% RSLogix 500 project MLO3B JOb 8.RSS, saved by version 10.00.00.00 %
PROJECT "MLO3B"    % processor: Bul.1763 MicroLogix 1100 Series B %

PROGRAM FILES
  LAD 2   5 rungs

DATA FILES
  O0 OUTPUT  4 elements
  I1 INPUT  6 elements
  S2 STATUS  66 elements
  B3 BINARY  1 elements
  T4 TIMER  1 elements
  C5 COUNTER  1 elements
  R6 CONTROL  1 elements
  N7 INTEGER  1 elements
  F8 FLOAT  1 elements

LADDER 2
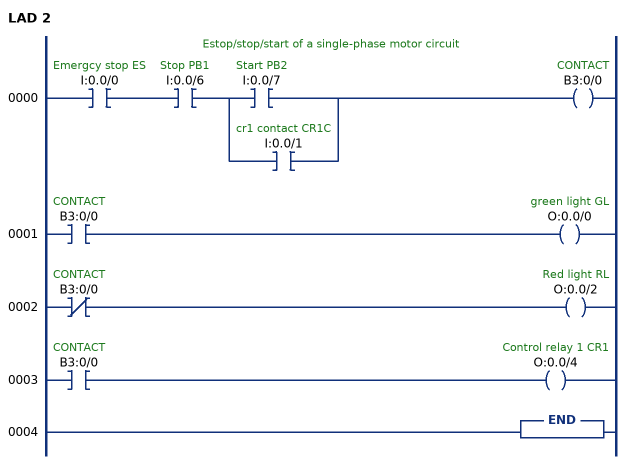
% Rung: 0 %
% Estop/stop/start of a single-phase motor circuit %
SOR XIC I:0.0/0 XIC I:0.0/6 BST XIC I:0.0/7 NXB XIC I:0.0/1 BND OTE B3:0/0 EOR
%   I:0.0/0  ES  "Emergcy stop" %
%   I:0.0/6  PB1  "Stop" %
%   I:0.0/7  PB2  "Start" %
%   I:0.0/1  CR1C  "cr1 contact" %
%   B3:0/0  CONTACT %
% Rung: 1 %
SOR XIC B3:0/0 OTE O:0.0/0 EOR
%   B3:0/0  CONTACT %
%   O:0.0/0  GL  "green light" %
% Rung: 2 %
SOR XIO B3:0/0 OTE O:0.0/2 EOR
%   B3:0/0  CONTACT %
%   O:0.0/2  RL  "Red light" %
% Rung: 3 %
SOR XIC B3:0/0 OTE O:0.0/4 EOR
%   B3:0/0  CONTACT %
%   O:0.0/4  CR1  "Control relay 1" %
% Rung: 4 %
SOR END EOR

OTHER DOCUMENTED ADDRESSES
  I:0.0/2  CR2C  "Start"
  I:0.0/3  3PSSA  "Three position selector switch a position"
  I:0.0/4  3PSSB  "Three postion selector switch b"
  I:0.0/5  2PSS  "Two postion selector switch"
  I:0.0/8  PB3  "Normaly open pushbutton"
  IOS  
  O:0.0/1  YL  "Yellow light"
  O:0.0/3  BL  "Blue light"
  O:0.0/5  CR2  "Control relay 2"
  O:0.0/6  RED_LIGHT
  O:0.0/7  "Green light"
